// Shift data from end to begin
FUNCTION ShiftDataLeft : BOOL
VAR_INPUT
	data : ANY;
	byteCount : UDINT; // How far to the left are shifted
END_VAR

MEMMOVE(destAddr := data.pValue, srcAddr := data.pValue + byteCount, n := TO_UDINT(data.diSize) - byteCount);
MEMSET(destAddr := data.pValue + TO_UDINT(data.diSize) - byteCount, fillByte := 0, n := byteCount);

END_FUNCTION

(* stored: Version 1.1.0.1
   POU ShiftDataLeft: Id {e97f8ec7-a46d-05b0-3d60-c70782600e15}, SpecialFunc None *)
